(* CoDeSys 2.3 export: ALL.EXP *)
(* Libraries: ANALYZATION.LIB 5.10.99 09:05:06, ComService.lib 21.5.09 14:28:28, IECSFC.LIB 13.4.06 15:51:28, modbus.lib 11.2.26 05:01:17, STANDARD.LIB 4.10.05 11:14:46, SysLibCom.lib 20.2.06 12:31:08 *)

(* PLC configuration (modules and I/O channels)
PLC110_30 [Root] node -1, in %IB0 out %QB0 {param 1 = PLC110-30_v2; param 2 = 1; param 3 = 1000}
  Fast discrete inputs [I_SIMPLE_INPUT] node 0, in %IB0 out %QB0 {param 1 = Fast discrete inputs; param 2 = 10000}
    AT %IX0.0 [BitInput] Дискретный вход 1 {param 1 = Enter name}
    AT %IX0.1 [BitInput] Дискретный вход 2 {param 1 = Enter name}
  Дискретные входы - 16 [ID130] node 1, in %IB1 out %QB1 {param 1 = Дискретные входы; param 2 = 10; param 3 = 16}
    AT %IB1.0 [ByteInput] 8 дискретных входов {param 1 = Enter name}
    AT %IB1.1 [ByteInput] 8 дискретных входов {param 1 = Enter name}
  Быстрые дискретные выходы [OWEN_ID570] node 2, in %IB2 out %QB2 {param 1 = Быстрые дискретные выходы; param 2 = FALSE; param 3 = FALSE; param 4 = FALSE; param 5 = FALSE}
    AT %QX2.0 [BitOutput] Быстрый дискретный выход 1 {param 1 = Enter name}
    AT %QX2.1 [BitOutput] Быстрый дискретный выход 2 {param 1 = Enter name}
    AT %QX2.2 [BitOutput] Быстрый дискретный выход 3 {param 1 = Enter name}
    AT %QX2.3 [BitOutput] Быстрый дискретный выход 4 {param 1 = Enter name}
  Дискретные выходы - 8 [ID131] node 3, in %IB3 out %QB3 {param 1 = Дискретные выходы; param 2 = 0; param 3 = No; param 4 = 10}
    AT %QB3.0 [ByteOutput] 8 дискретных выходов {param 1 = Enter name}
  Специальный вход [ID103] node 4, in %IB4 out %QB4 {param 1 = Специальный вход}
    AT %IX4.0 [BitInput] Специальный вход {param 1 = Enter name}
  Специальный выход [ID104] node 5, in %IB5 out %QB5 {param 1 = Специальный выход}
    AT %QX5.0 [BitOutput] Специальный выход {param 1 = Enter name}
  ModBus (Master) [MODBUS_MASTER_ID450] node 6, in %IB6 out %QB6 {param 1 = ModBus (Master); param 2 = No}
    AT %QD6.0 [DWordOutput] Last address {param 1 = Enter name}
    AT %QW6.1 [WordOutput] Last error {param 1 = Enter name}
    RS-485-1 [COM1_USART] node 0, in %IB6.0 out %QB6.0 {param 1 = RS-485-1; param 2 = 9600; param 3 = NO PARITY CHECK; param 4 = 8 bits; param 5 = One stop bit; param 6 = RS485; param 7 = ASCII; param 8 = 0; param 9 = No}
*)

(* Global variable list: Global_Variables *)
VAR_GLOBAL
    (* Fast discrete inputs (encoder) *)
    gEncoderA   AT %IX0.0 : BOOL;    (* DI1 - Encoder A (fast input) *)
    gEncoderB   AT %IX0.1 : BOOL;    (* DI2 - Encoder B (fast input) *)

    (* ModBus (Master) system/channel variables exposed by device configuration *)
    gModbus_Master_Channel AT %QD6.0 : DWORD; (* ModBus Master: channel/last address (Q area) *)
    gModbus_Master_LastError AT %QW6.1 : WORD; (* ModBus Master: last error code (Q area) *)

    (* Discrete inputs (DI3..DI18) mapped to %IX1.0.0 - %IX1.1.7 *)
    gDI_3  AT %IX1.0.0 : BOOL; (* DI3 *)
    gDI_4  AT %IX1.0.1 : BOOL; (* DI4 *)
    gDI_5  AT %IX1.0.2 : BOOL; (* DI5 *)
    gDI_6  AT %IX1.0.3 : BOOL; (* DI6 *)
    gDI_7  AT %IX1.0.4 : BOOL; (* DI7 *)
    gDI_8  AT %IX1.0.5 : BOOL; (* DI8 *)
    gDI_9  AT %IX1.0.6 : BOOL; (* DI9 *)
    gDI_10 AT %IX1.0.7 : BOOL; (* DI10 *)
    gDI_11 AT %IX1.1.0 : BOOL; (* DI11 *)
    gDI_12 AT %IX1.1.1 : BOOL; (* DI12 *)
    gDI_13 AT %IX1.1.2 : BOOL; (* DI13 *)
    gDI_14 AT %IX1.1.3 : BOOL; (* DI14 *)
    gDI_15 AT %IX1.1.4 : BOOL; (* DI15 *)
    gDI_16 AT %IX1.1.5 : BOOL; (* DI16 *)
    gDI_17 AT %IX1.1.6 : BOOL; (* DI17 *)
    gDI_18 AT %IX1.1.7 : BOOL; (* DI18 *)

    (* Discrete outputs - relay DO1..DO8 mapped to %QX3.0.0..%QX3.0.7 *)
    gDO_1 AT %QX3.0.0 : BOOL;  (* DO1 - Forward *)
    gDO_2 AT %QX3.0.1 : BOOL;  (* DO2 - Reverse *)
    gDO_3 AT %QX3.0.2 : BOOL;  (* DO3 - In position indicator *)
    gDO_4 AT %QX3.0.3 : BOOL;  (* DO4 *)
    gDO_5 AT %QX3.0.4 : BOOL;  (* DO5 *)
    gDO_6 AT %QX3.0.5 : BOOL;  (* DO6 *)
    gDO_7 AT %QX3.0.6 : BOOL;  (* DO7 *)
    gDO_8 AT %QX3.0.7 : BOOL;  (* DO8 *)

    (* Fast/transistor discrete outputs DO9..DO12 mapped to %QX2.0..%QX2.3 (fast outputs module) *)
    gDO_9  AT %QX2.0 : BOOL; (* DO9  - fast/transistor output *)
    gDO_10 AT %QX2.1 : BOOL; (* DO10 *)
    gDO_11 AT %QX2.2 : BOOL; (* DO11 *)
    gDO_12 AT %QX2.3 : BOOL; (* DO12 *)

    (* Variables for Modbus and internal state (no AT) *)
    (*
        Modbus (holding) register map served by ESP (slave):
        Register numbers (offset 0):
        0-1   : target angle (REAL)            (REG_TARGET_ANGLE_HI/LO)
        2-3   : current angle (REAL)           (REG_CURRENT_ANGLE_HI/LO)
        4-5   : reserved
        6     : status (WORD)                  (0=Stop,1=Moving,2=In position)
        7     : error code (WORD)
        8     : command (WORD)                 (1=Start,2=Stop,3=Calib)
        9-10  : encoder count (DINT, hi/lo)
        11    : PPR (WORD)
        12    : quad mode (WORD)
        13    : max time (WORD)
        14-15 : hysteresis (REAL)
    *)
    gTargetAngle : REAL := 45.0;    (* target angle, degrees *)
    gCurrentAngle : REAL := 0.0;    (* current angle, degrees *)
    gAngleFromStart : REAL := 0.0;  (* angle from program start *)
    gStatus : INT := 0;             (* 0=Stop,1=Moving,2=In position *)
    gErrorCode : INT := 0;          (* 0=OK,1=Timeout,2=Fault *)
    gCommand : INT := 0;            (* 1=Start,2=Stop,3=Calibrate *)
    gEncoderCount : DINT := 0;     (* encoder counter for Modbus *)

    (* Calibration / Modbus helper variables *)
    gStartCalib : BOOL := FALSE;
    gCalibRunning : BOOL := FALSE;
    gCalibStatus : INT := 0;
    gCalibRevsDone : INT := 0;
    gCalibRevsTarget : INT := 3;
    gCalibMeasured : REAL := 0.0;
    gCalibCountsPerRev : DINT := 0;
END_VAR

(* POU PLC_PRG, ST *)
(* COMSETTINGS type usage is handled inside program files; fallback type removed here to avoid duplicate definition. If needed, define COMSETTINGS or COMSETTINGS_FALLBACK inside the POU file that uses it (e.g., `all2.exp`). *)
PROGRAM PLC_PRG
VAR
    COUNTS_PER_REV : INT := 360;
    ANGLE_PER_COUNT : REAL := 1.0;
    HYSTERESIS : REAL := 1.5;
    MAX_MOVE_TIME : INT := 3000;
    encoderCount : DINT := 0;
    zeroOffset : DINT := 0;
    moveTimer : INT := 0;
    isMoving : BOOL := FALSE;
    isPositioned : BOOL := FALSE;
    prevCalibBtn : BOOL := FALSE;
    prevEncoderA : BOOL := FALSE;
    startOffset : DINT := 0;
    started : BOOL := FALSE;
    tmpAngle : REAL := 0.0;
    tmpStartAngle : REAL := 0.0;
    tmpTarget : REAL := 0.0;
    tmpDiff : REAL := 0.0;
    motorFwd : BOOL := FALSE;
    motorRev : BOOL := FALSE;
    calibBtn : BOOL := FALSE;
    motorEnable : BOOL := FALSE;
    alarmInput : BOOL := FALSE;
    allDOBtn : BOOL := FALSE;
    mbRes : INT;
    mbBuf : ARRAY[0..15] OF WORD;
    dw : DWORD;
    tmpReal : REAL;
END_VAR
calibBtn := gDI_7;
motorEnable := gDI_8;
alarmInput := gDI_9;

IF gEncoderA AND NOT prevEncoderA THEN
    IF gEncoderB THEN
        encoderCount := encoderCount - 1;
    ELSE
        encoderCount := encoderCount + 1;
    END_IF;
END_IF;
IF NOT gEncoderA AND prevEncoderA THEN
    IF gEncoderB THEN
        encoderCount := encoderCount + 1;
    ELSE
        encoderCount := encoderCount - 1;
    END_IF;
END_IF;
prevEncoderA := gEncoderA;

gEncoderCount := encoderCount;

gCurrentAngle := DINT_TO_REAL((encoderCount MOD 360 + 360) MOD 360) * ANGLE_PER_COUNT;

tmpTarget := gTargetAngle;
WHILE tmpTarget < 0.0 DO
    tmpTarget := tmpTarget + 360.0;
END_WHILE;
WHILE tmpTarget >= 360.0 DO
    tmpTarget := tmpTarget - 360.0;
END_WHILE;

tmpDiff := tmpTarget - gCurrentAngle;
IF tmpDiff > 180.0 THEN
    tmpDiff := tmpDiff - 360.0;
ELSIF tmpDiff < -180.0 THEN
    mbRes := -1;
    tmpDiff := tmpDiff + 360.0;
END_IF;

IF alarmInput THEN
    motorFwd := FALSE;
    motorRev := FALSE;
    isMoving := FALSE;
    gErrorCode := 2;
    gStatus := 0;
END_IF;

IF motorEnable AND NOT alarmInput AND (gCommand <> 2) THEN
    IF ABS(tmpDiff) <= HYSTERESIS THEN
        motorFwd := FALSE;
        motorRev := FALSE;
        isPositioned := TRUE;
        isMoving := FALSE;
        moveTimer := 0;
        gStatus := 2;
        IF gErrorCode = 1 THEN
            gErrorCode := 0;
        END_IF;
    ELSE
        isPositioned := FALSE;
        isMoving := TRUE;
        gStatus := 1;
        IF tmpDiff > 0.0 THEN
            motorFwd := TRUE;
            motorRev := FALSE;
        ELSE
            motorFwd := FALSE;
            motorRev := TRUE;
        END_IF;
        moveTimer := moveTimer + 1;
        IF moveTimer > MAX_MOVE_TIME THEN
            motorFwd := FALSE;
            motorRev := FALSE;
            isMoving := FALSE;
            gErrorCode := 1;
            gStatus := 0;
        END_IF;
    END_IF;
ELSE
    motorFwd := FALSE;
    motorRev := FALSE;
    isMoving := FALSE;
    IF NOT alarmInput THEN
        gStatus := 0;
    END_IF;
END_IF;

IF gCommand = 2 THEN
    motorFwd := FALSE;
    motorRev := FALSE;
    isMoving := FALSE;
    gStatus := 0;
END_IF;

allDOBtn := gDI_7;
IF allDOBtn THEN
    gDO_1 := TRUE;
    gDO_2 := TRUE;
    gDO_3 := TRUE;
    gDO_4 := TRUE;
    gDO_5 := TRUE;
    gDO_6 := TRUE;
    gDO_7 := TRUE;
    gDO_8 := TRUE;
ELSE
    gDO_1 := motorFwd;
    gDO_2 := motorRev;
    gDO_3 := isPositioned;
END_IF;
END_PROGRAM
